// TIA Portal V15.1 export
// export: Created 2020-06-12T07:35:48.8818359Z, ExportSetting None, DisplayName Totally Integrated Automation Portal, DisplayVersion V15.1, DisplayName TIA Portal Openness, DisplayVersion V15.1, DisplayName STEP 7 Professional, DisplayVersion V15.1, DisplayName STEP 7 Safety, DisplayVersion V15.1, DisplayName WinCC Advanced, DisplayVersion V15.1
FUNCTION "XY_call" : Void   // FC84, FBD
TITLE = XY-adjustment call
{ S7_Optimized_Access := 'TRUE' }
// stored: SetENOAutomatically False
BEGIN

REGION Network 1: XY Movement
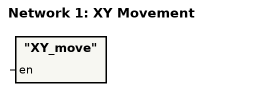
   "XY_move"();
END_REGION
END_FUNCTION
